(* PLC project SafeLOGIC-1, BrAutomation SafeDESIGNER  4.2.0.17 *)
(* stored: companyURL http://www.br-automation.com, creationDateTime Thu Sep 08 10:43:09 2016 *)

PROGRAM Main

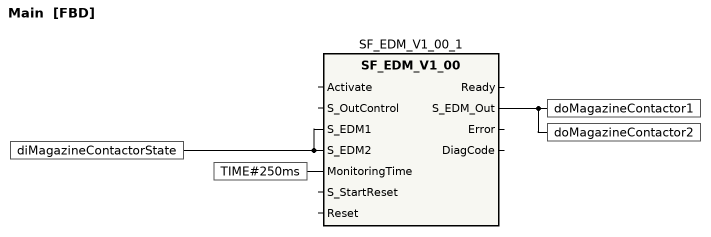
(* FBD diagram, written out as Structured Text *)
SF_EDM_V1_00_1(S_EDM1 := diMagazineContactorState, S_EDM2 := diMagazineContactorState, MonitoringTime := TIME#250ms);
doMagazineContactor2 := SF_EDM_V1_00_1.S_EDM_Out;
doMagazineContactor1 := SF_EDM_V1_00_1.S_EDM_Out;
END_PROGRAM
